# EPICS substitutions: ioc/iocBoot/iocsm/Db/backup/galil_digital_ports.substitutions
# Description:
# digital/binary port substitution file.
#
# This library is free software; you can redistribute it and/or
# modify it under the terms of the GNU Lesser General Public
# Licence as published by the Free Software Foundation; either
# version 2.1 of the Licence, or (at your option) any later version.
#
# This library is distributed in the hope that it will be useful,
# but WITHOUT ANY WARRANTY; without even the implied warranty of
# MERCHANTABILITY or FITNESS FOR A PARTICULAR PURPOSE.  See the GNU
# Lesser General Public Licence for more details.
#
# You should have received a copy of the GNU Lesser General Public
# Licence along with this library; if not, write to the Free Software
# Foundation, Inc., 51 Franklin St, Fifth Floor, Boston, MA 02110-1301 USA.
#
# Contact details:
# mark.clift@synchrotron.org.au
# 800 Blackburn Road, Clayton, Victoria 3168, Australia.
#

# P    - PV prefix
# R    - Record Name
# PORT - Asyn port name
# BYTE - Hardware byte to read
# MASK - Mask for this bit

file "$(GALIL)/GalilSup/Db/galil_digital_in_bit.template"
{
pattern {P,      R,          PORT,  BYTE,  MASK,     ZNAM,  ONAM,  ZSV,        OSV         }

	{X14B1:EX,  Galil0Bi0,  Galil2183, 0,     0x000001, "Off", "On",  "NO_ALARM", "NO_ALARM"  }
	{X14B1:EX,  Galil0Bi1,  Galil2183, 0,     0x000002, "Off", "On",  "NO_ALARM", "NO_ALARM"  }
	{X14B1:EX,  Galil0Bi2,  Galil2183, 0,     0x000004, "Off", "On",  "NO_ALARM", "NO_ALARM"  }
	{X14B1:EX,  Galil0Bi3,  Galil2183, 0,     0x000008, "Off", "On",  "NO_ALARM", "NO_ALARM"  }
	{X14B1:EX,  Galil0Bi4,  Galil2183, 0,     0x000010, "Off", "On",  "NO_ALARM", "NO_ALARM"  }
	{X14B1:EX,  Galil0Bi5,  Galil2183, 0,     0x000020, "Off", "On",  "NO_ALARM", "NO_ALARM"  }
	{X14B1:EX,  Galil0Bi6,  Galil2183, 0,     0x000040, "Off", "On",  "NO_ALARM", "NO_ALARM"  }
	{X14B1:EX,  Galil0Bi7,  Galil2183, 0,     0x000080, "Off", "On",  "NO_ALARM", "NO_ALARM"  }

	{X14B1:EX,  Galil1Bi0,  Galil2183, 1,     0x000001, "Off", "On",  "NO_ALARM", "NO_ALARM"  }
	{X14B1:EX,  Galil1Bi1,  Galil2183, 1,     0x000002, "Off", "On",  "NO_ALARM", "NO_ALARM"  }
	{X14B1:EX,  Galil1Bi2,  Galil2183, 1,     0x000004, "Off", "On",  "NO_ALARM", "NO_ALARM"  }
	{X14B1:EX,  Galil1Bi3,  Galil2183, 1,     0x000008, "Off", "On",  "NO_ALARM", "NO_ALARM"  }
	{X14B1:EX,  Galil1Bi4,  Galil2183, 1,     0x000010, "Off", "On",  "NO_ALARM", "NO_ALARM"  }
	{X14B1:EX,  Galil1Bi5,  Galil2183, 1,     0x000020, "Off", "On",  "NO_ALARM", "NO_ALARM"  }
	{X14B1:EX,  Galil1Bi6,  Galil2183, 1,     0x000040, "Off", "On",  "NO_ALARM", "NO_ALARM"  }
	{X14B1:EX,  Galil1Bi7,  Galil2183, 1,     0x000080, "Off", "On",  "NO_ALARM", "NO_ALARM"  }

	{X14B1:EX,  Galil2Bi0,  Galil2183, 2,     0x000001, "Off", "On",  "NO_ALARM", "NO_ALARM"  }
	{X14B1:EX,  Galil2Bi1,  Galil2183, 2,     0x000002, "Off", "On",  "NO_ALARM", "NO_ALARM"  }
	{X14B1:EX,  Galil2Bi2,  Galil2183, 2,     0x000004, "Off", "On",  "NO_ALARM", "NO_ALARM"  }
	{X14B1:EX,  Galil2Bi3,  Galil2183, 2,     0x000008, "Off", "On",  "NO_ALARM", "NO_ALARM"  }
	{X14B1:EX,  Galil2Bi4,  Galil2183, 2,     0x000010, "Off", "On",  "NO_ALARM", "NO_ALARM"  }
	{X14B1:EX,  Galil2Bi5,  Galil2183, 2,     0x000020, "Off", "On",  "NO_ALARM", "NO_ALARM"  }
	{X14B1:EX,  Galil2Bi6,  Galil2183, 2,     0x000040, "Off", "On",  "NO_ALARM", "NO_ALARM"  }
	{X14B1:EX,  Galil2Bi7,  Galil2183, 2,     0x000080, "Off", "On",  "NO_ALARM", "NO_ALARM"  }

	{X14B1:EX,  Galil3Bi0,  Galil2183, 3,     0x000001, "Off", "On",  "NO_ALARM", "NO_ALARM"  }
	{X14B1:EX,  Galil3Bi1,  Galil2183, 3,     0x000002, "Off", "On",  "NO_ALARM", "NO_ALARM"  }
	{X14B1:EX,  Galil3Bi2,  Galil2183, 3,     0x000004, "Off", "On",  "NO_ALARM", "NO_ALARM"  }
	{X14B1:EX,  Galil3Bi3,  Galil2183, 3,     0x000008, "Off", "On",  "NO_ALARM", "NO_ALARM"  }
	{X14B1:EX,  Galil3Bi4,  Galil2183, 3,     0x000010, "Off", "On",  "NO_ALARM", "NO_ALARM"  }
	{X14B1:EX,  Galil3Bi5,  Galil2183, 3,     0x000020, "Off", "On",  "NO_ALARM", "NO_ALARM"  }
	{X14B1:EX,  Galil3Bi6,  Galil2183, 3,     0x000040, "Off", "On",  "NO_ALARM", "NO_ALARM"  }
	{X14B1:EX,  Galil3Bi7,  Galil2183, 3,     0x000080, "Off", "On",  "NO_ALARM", "NO_ALARM"  }

	{X14B1:EX,  Galil4Bi0,  Galil2183, 4,     0x000001, "Off", "On",  "NO_ALARM", "NO_ALARM"  }
	{X14B1:EX,  Galil4Bi1,  Galil2183, 4,     0x000002, "Off", "On",  "NO_ALARM", "NO_ALARM"  }
	{X14B1:EX,  Galil4Bi2,  Galil2183, 4,     0x000004, "Off", "On",  "NO_ALARM", "NO_ALARM"  }
	{X14B1:EX,  Galil4Bi3,  Galil2183, 4,     0x000008, "Off", "On",  "NO_ALARM", "NO_ALARM"  }
	{X14B1:EX,  Galil4Bi4,  Galil2183, 4,     0x000010, "Off", "On",  "NO_ALARM", "NO_ALARM"  }
	{X14B1:EX,  Galil4Bi5,  Galil2183, 4,     0x000020, "Off", "On",  "NO_ALARM", "NO_ALARM"  }
	{X14B1:EX,  Galil4Bi6,  Galil2183, 4,     0x000040, "Off", "On",  "NO_ALARM", "NO_ALARM"  }
	{X14B1:EX,  Galil4Bi7,  Galil2183, 4,     0x000080, "Off", "On",  "NO_ALARM", "NO_ALARM"  }

	{X14B1:EX,  Galil5Bi0,  Galil2183, 5,     0x000001, "Off", "On",  "NO_ALARM", "NO_ALARM"  }
	{X14B1:EX,  Galil5Bi1,  Galil2183, 5,     0x000002, "Off", "On",  "NO_ALARM", "NO_ALARM"  }
	{X14B1:EX,  Galil5Bi2,  Galil2183, 5,     0x000004, "Off", "On",  "NO_ALARM", "NO_ALARM"  }
	{X14B1:EX,  Galil5Bi3,  Galil2183, 5,     0x000008, "Off", "On",  "NO_ALARM", "NO_ALARM"  }
	{X14B1:EX,  Galil5Bi4,  Galil2183, 5,     0x000010, "Off", "On",  "NO_ALARM", "NO_ALARM"  }
	{X14B1:EX,  Galil5Bi5,  Galil2183, 5,     0x000020, "Off", "On",  "NO_ALARM", "NO_ALARM"  }
	{X14B1:EX,  Galil5Bi6,  Galil2183, 5,     0x000040, "Off", "On",  "NO_ALARM", "NO_ALARM"  }
	{X14B1:EX,  Galil5Bi7,  Galil2183, 5,     0x000080, "Off", "On",  "NO_ALARM", "NO_ALARM"  }

	{X14B1:EX,  Galil6Bi0,  Galil2183, 6,     0x000001, "Off", "On",  "NO_ALARM", "NO_ALARM"  }
	{X14B1:EX,  Galil6Bi1,  Galil2183, 6,     0x000002, "Off", "On",  "NO_ALARM", "NO_ALARM"  }
	{X14B1:EX,  Galil6Bi2,  Galil2183, 6,     0x000004, "Off", "On",  "NO_ALARM", "NO_ALARM"  }
	{X14B1:EX,  Galil6Bi3,  Galil2183, 6,     0x000008, "Off", "On",  "NO_ALARM", "NO_ALARM"  }
	{X14B1:EX,  Galil6Bi4,  Galil2183, 6,     0x000010, "Off", "On",  "NO_ALARM", "NO_ALARM"  }
	{X14B1:EX,  Galil6Bi5,  Galil2183, 6,     0x000020, "Off", "On",  "NO_ALARM", "NO_ALARM"  }
	{X14B1:EX,  Galil6Bi6,  Galil2183, 6,     0x000040, "Off", "On",  "NO_ALARM", "NO_ALARM"  }
	{X14B1:EX,  Galil6Bi7,  Galil2183, 6,     0x000080, "Off", "On",  "NO_ALARM", "NO_ALARM"  }

# RIO binary inputs are organized in bytes

}

# P    - PV prefix
# R    - Record Name
# PORT - Asyn port name
# WORD - Hardware word to read
# MASK - Mask for this bit

file "$(GALIL)/GalilSup/Db/galil_digital_out_bit.template"
{
pattern {P,      R,           PORT,  WORD,  MASK,     ZNAM,  ONAM,  ZSV,        OSV         }

# DMC binary outputs are organized in 16bit words
	{X14B1:EX,  Galil0Bo0,   Galil2183, 0,     0x000001, "Off", "On",  "NO_ALARM", "NO_ALARM"  }
	{X14B1:EX,  Galil0Bo1,   Galil2183, 0,     0x000002, "Off", "On",  "NO_ALARM", "NO_ALARM"  }
	{X14B1:EX,  Galil0Bo2,   Galil2183, 0,     0x000004, "Off", "On",  "NO_ALARM", "NO_ALARM"  }
	{X14B1:EX,  Galil0Bo3,   Galil2183, 0,     0x000008, "Off", "On",  "NO_ALARM", "NO_ALARM"  }
	{X14B1:EX,  Galil0Bo4,   Galil2183, 0,     0x000010, "Off", "On",  "NO_ALARM", "NO_ALARM"  }
	{X14B1:EX,  Galil0Bo5,   Galil2183, 0,     0x000020, "Off", "On",  "NO_ALARM", "NO_ALARM"  }
	{X14B1:EX,  Galil0Bo6,   Galil2183, 0,     0x000040, "Off", "On",  "NO_ALARM", "NO_ALARM"  }
	{X14B1:EX,  Galil0Bo7,   Galil2183, 0,     0x000080, "Off", "On",  "NO_ALARM", "NO_ALARM"  }
	{X14B1:EX,  Galil0Bo8,   Galil2183, 0,     0x000100, "Off", "On",  "NO_ALARM", "NO_ALARM"  }
	{X14B1:EX,  Galil0Bo9,   Galil2183, 0,     0x000200, "Off", "On",  "NO_ALARM", "NO_ALARM"  }
	{X14B1:EX,  Galil0Bo10,  Galil2183, 0,     0x000400, "Off", "On",  "NO_ALARM", "NO_ALARM"  }
	{X14B1:EX,  Galil0Bo11,  Galil2183, 0,     0x000800, "Off", "On",  "NO_ALARM", "NO_ALARM"  }
	{X14B1:EX,  Galil0Bo12,  Galil2183, 0,     0x001000, "Off", "On",  "NO_ALARM", "NO_ALARM"  }
	{X14B1:EX,  Galil0Bo13,  Galil2183, 0,     0x002000, "Off", "On",  "NO_ALARM", "NO_ALARM"  }
	{X14B1:EX,  Galil0Bo14,  Galil2183, 0,     0x004000, "Off", "On",  "NO_ALARM", "NO_ALARM"  }
	{X14B1:EX,  Galil0Bo15,  Galil2183, 0,     0x008000, "Off", "On",  "NO_ALARM", "NO_ALARM"  }

	{X14B1:EX,  Galil1Bo0,   Galil2183, 1,     0x000001, "Off", "On",  "NO_ALARM", "NO_ALARM"  }
	{X14B1:EX,  Galil1Bo1,   Galil2183, 1,     0x000002, "Off", "On",  "NO_ALARM", "NO_ALARM"  }
	{X14B1:EX,  Galil1Bo2,   Galil2183, 1,     0x000004, "Off", "On",  "NO_ALARM", "NO_ALARM"  }
	{X14B1:EX,  Galil1Bo3,   Galil2183, 1,     0x000008, "Off", "On",  "NO_ALARM", "NO_ALARM"  }
	{X14B1:EX,  Galil1Bo4,   Galil2183, 1,     0x000010, "Off", "On",  "NO_ALARM", "NO_ALARM"  }
	{X14B1:EX,  Galil1Bo5,   Galil2183, 1,     0x000020, "Off", "On",  "NO_ALARM", "NO_ALARM"  }
	{X14B1:EX,  Galil1Bo6,   Galil2183, 1,     0x000040, "Off", "On",  "NO_ALARM", "NO_ALARM"  }
	{X14B1:EX,  Galil1Bo7,   Galil2183, 1,     0x000080, "Off", "On",  "NO_ALARM", "NO_ALARM"  }
	{X14B1:EX,  Galil1Bo8,   Galil2183, 1,     0x000100, "Off", "On",  "NO_ALARM", "NO_ALARM"  }
	{X14B1:EX,  Galil1Bo9,   Galil2183, 1,     0x000200, "Off", "On",  "NO_ALARM", "NO_ALARM"  }
	{X14B1:EX,  Galil1Bo10,  Galil2183, 1,     0x000400, "Off", "On",  "NO_ALARM", "NO_ALARM"  }
	{X14B1:EX,  Galil1Bo11,  Galil2183, 1,     0x000800, "Off", "On",  "NO_ALARM", "NO_ALARM"  }
	{X14B1:EX,  Galil1Bo12,  Galil2183, 1,     0x001000, "Off", "On",  "NO_ALARM", "NO_ALARM"  }
	{X14B1:EX,  Galil1Bo13,  Galil2183, 1,     0x002000, "Off", "On",  "NO_ALARM", "NO_ALARM"  }
	{X14B1:EX,  Galil1Bo14,  Galil2183, 1,     0x004000, "Off", "On",  "NO_ALARM", "NO_ALARM"  }
	{X14B1:EX,  Galil1Bo15,  Galil2183, 1,     0x008000, "Off", "On",  "NO_ALARM", "NO_ALARM"  }

	{X14B1:EX,  Galil2Bo0,   Galil2183, 2,     0x000001, "Off", "On",  "NO_ALARM", "NO_ALARM"  }
	{X14B1:EX,  Galil2Bo1,   Galil2183, 2,     0x000002, "Off", "On",  "NO_ALARM", "NO_ALARM"  }
	{X14B1:EX,  Galil2Bo2,   Galil2183, 2,     0x000004, "Off", "On",  "NO_ALARM", "NO_ALARM"  }
	{X14B1:EX,  Galil2Bo3,   Galil2183, 2,     0x000008, "Off", "On",  "NO_ALARM", "NO_ALARM"  }
	{X14B1:EX,  Galil2Bo4,   Galil2183, 2,     0x000010, "Off", "On",  "NO_ALARM", "NO_ALARM"  }
	{X14B1:EX,  Galil2Bo5,   Galil2183, 2,     0x000020, "Off", "On",  "NO_ALARM", "NO_ALARM"  }
	{X14B1:EX,  Galil2Bo6,   Galil2183, 2,     0x000040, "Off", "On",  "NO_ALARM", "NO_ALARM"  }
	{X14B1:EX,  Galil2Bo7,   Galil2183, 2,     0x000080, "Off", "On",  "NO_ALARM", "NO_ALARM"  }
	{X14B1:EX,  Galil2Bo8,   Galil2183, 2,     0x000100, "Off", "On",  "NO_ALARM", "NO_ALARM"  }
	{X14B1:EX,  Galil2Bo9,   Galil2183, 2,     0x000200, "Off", "On",  "NO_ALARM", "NO_ALARM"  }
	{X14B1:EX,  Galil2Bo10,  Galil2183, 2,     0x000400, "Off", "On",  "NO_ALARM", "NO_ALARM"  }
	{X14B1:EX,  Galil2Bo11,  Galil2183, 2,     0x000800, "Off", "On",  "NO_ALARM", "NO_ALARM"  }
	{X14B1:EX,  Galil2Bo12,  Galil2183, 2,     0x001000, "Off", "On",  "NO_ALARM", "NO_ALARM"  }
	{X14B1:EX,  Galil2Bo13,  Galil2183, 2,     0x002000, "Off", "On",  "NO_ALARM", "NO_ALARM"  }
	{X14B1:EX,  Galil2Bo14,  Galil2183, 2,     0x004000, "Off", "On",  "NO_ALARM", "NO_ALARM"  }
	{X14B1:EX,  Galil2Bo15,  Galil2183, 2,     0x008000, "Off", "On",  "NO_ALARM", "NO_ALARM"  }

	{X14B1:EX,  Galil3Bo0,   Galil2183, 3,     0x000001, "Off", "On",  "NO_ALARM", "NO_ALARM"  }
	{X14B1:EX,  Galil3Bo1,   Galil2183, 3,     0x000002, "Off", "On",  "NO_ALARM", "NO_ALARM"  }
	{X14B1:EX,  Galil3Bo2,   Galil2183, 3,     0x000004, "Off", "On",  "NO_ALARM", "NO_ALARM"  }
	{X14B1:EX,  Galil3Bo3,   Galil2183, 3,     0x000008, "Off", "On",  "NO_ALARM", "NO_ALARM"  }
	{X14B1:EX,  Galil3Bo4,   Galil2183, 3,     0x000010, "Off", "On",  "NO_ALARM", "NO_ALARM"  }
	{X14B1:EX,  Galil3Bo5,   Galil2183, 3,     0x000020, "Off", "On",  "NO_ALARM", "NO_ALARM"  }
	{X14B1:EX,  Galil3Bo6,   Galil2183, 3,     0x000040, "Off", "On",  "NO_ALARM", "NO_ALARM"  }
	{X14B1:EX,  Galil3Bo7,   Galil2183, 3,     0x000080, "Off", "On",  "NO_ALARM", "NO_ALARM"  }
	{X14B1:EX,  Galil3Bo8,   Galil2183, 3,     0x000100, "Off", "On",  "NO_ALARM", "NO_ALARM"  }
	{X14B1:EX,  Galil3Bo9,   Galil2183, 3,     0x000200, "Off", "On",  "NO_ALARM", "NO_ALARM"  }
	{X14B1:EX,  Galil3Bo10,  Galil2183, 3,     0x000400, "Off", "On",  "NO_ALARM", "NO_ALARM"  }
	{X14B1:EX,  Galil3Bo11,  Galil2183, 3,     0x000800, "Off", "On",  "NO_ALARM", "NO_ALARM"  }
	{X14B1:EX,  Galil3Bo12,  Galil2183, 3,     0x001000, "Off", "On",  "NO_ALARM", "NO_ALARM"  }
	{X14B1:EX,  Galil3Bo13,  Galil2183, 3,     0x002000, "Off", "On",  "NO_ALARM", "NO_ALARM"  }
	{X14B1:EX,  Galil3Bo14,  Galil2183, 3,     0x004000, "Off", "On",  "NO_ALARM", "NO_ALARM"  }
	{X14B1:EX,  Galil3Bo15,  Galil2183, 3,     0x008000, "Off", "On",  "NO_ALARM", "NO_ALARM"  }

	{X14B1:EX,  Galil4Bo0,   Galil2183, 4,     0x000001, "Off", "On",  "NO_ALARM", "NO_ALARM"  }
	{X14B1:EX,  Galil4Bo1,   Galil2183, 4,     0x000002, "Off", "On",  "NO_ALARM", "NO_ALARM"  }
	{X14B1:EX,  Galil4Bo2,   Galil2183, 4,     0x000004, "Off", "On",  "NO_ALARM", "NO_ALARM"  }
	{X14B1:EX,  Galil4Bo3,   Galil2183, 4,     0x000008, "Off", "On",  "NO_ALARM", "NO_ALARM"  }
	{X14B1:EX,  Galil4Bo4,   Galil2183, 4,     0x000010, "Off", "On",  "NO_ALARM", "NO_ALARM"  }
	{X14B1:EX,  Galil4Bo5,   Galil2183, 4,     0x000020, "Off", "On",  "NO_ALARM", "NO_ALARM"  }
	{X14B1:EX,  Galil4Bo6,   Galil2183, 4,     0x000040, "Off", "On",  "NO_ALARM", "NO_ALARM"  }
	{X14B1:EX,  Galil4Bo7,   Galil2183, 4,     0x000080, "Off", "On",  "NO_ALARM", "NO_ALARM"  }
	{X14B1:EX,  Galil4Bo8,   Galil2183, 4,     0x000100, "Off", "On",  "NO_ALARM", "NO_ALARM"  }
	{X14B1:EX,  Galil4Bo9,   Galil2183, 4,     0x000200, "Off", "On",  "NO_ALARM", "NO_ALARM"  }
	{X14B1:EX,  Galil4Bo10,  Galil2183, 4,     0x000400, "Off", "On",  "NO_ALARM", "NO_ALARM"  }
	{X14B1:EX,  Galil4Bo11,  Galil2183, 4,     0x000800, "Off", "On",  "NO_ALARM", "NO_ALARM"  }
	{X14B1:EX,  Galil4Bo12,  Galil2183, 4,     0x001000, "Off", "On",  "NO_ALARM", "NO_ALARM"  }
	{X14B1:EX,  Galil4Bo13,  Galil2183, 4,     0x002000, "Off", "On",  "NO_ALARM", "NO_ALARM"  }
	{X14B1:EX,  Galil4Bo14,  Galil2183, 4,     0x004000, "Off", "On",  "NO_ALARM", "NO_ALARM"  }
	{X14B1:EX,  Galil4Bo15,  Galil2183, 4,     0x008000, "Off", "On",  "NO_ALARM", "NO_ALARM"  }

}

# end
